# EPICS autosave request: support/quadEM-2-4-1/quadEMApp/Db/quadEM_settings.req
# FILE... quadEM_settings.req
$(P)$(EM)Offset1
$(P)$(EM)Offset2
$(P)$(EM)Offset3
$(P)$(EM)Offset4
$(P)$(EM)PingPong1
$(P)$(EM)PingPong2
$(P)$(EM)PingPong3
$(P)$(EM)PingPong4
$(P)$(EM)ConversionTime
$(P)$(EM)Gain
$(P)$(EM)Read.SCAN
